TYPE ST_PNOutput_DCCharger :
STRUCT
	statusbits		:	DWORD;
	ChargerStatus	:	DWORD;
	ChargePower		:	DWORD;
END_STRUCT
END_TYPE

(* stored: Version 1.1.0.1, ProductVersion 3.1.4024.12
   DUT ST_PNOutput_DCCharger: Id {da3c5c79-3dde-4f5e-bb2e-d037ea22b5d2} *)
